{attribute 'reflection'}
FUNCTION_BLOCK FB_DevKL5151 EXTENDS FB_DevBase IMPLEMENTS iCounter
VAR_INPUT
	bInitAsCounterCard	: BOOL := FALSE; // (Default = FALSE) Use Terminal as encoder input (FALSE) or counter (TRUE) 
END_VAR
VAR CONSTANT // register values 
	WRITE_FEATURE_REGISTER 	: USINT := 16#E0; // write to register address command
	READ_FEATURE_REGISTER	: USINT := 16#A0; // Read feature register response  
END_VAR
VAR // Inputs and outputs
	Status		AT%I* : USINT ; // status byte from card
	Counter		AT%I* : UDINT ; // 
	Ctrl 		AT%Q* : USINT ; // Control byte to card`
	DataOut 	AT%Q* : UDINT ; // Set counter value
END_VAR
VAR // steppers
	InitStep : INT := 0; // init stepper
END_VAR
VAR // Manual control
	stManualControl : st_ManualCounterControl;
END_VAR

SUPER^();

METHOD PUBLIC CmdManual : BOOL
bCmdManual := TRUE;
stManualControl.nCount := Counter;

IF stManualControl.bManSetValue THEN 
	// set counter to value
	DataOut	:= stManualControl.nManValue	;
	Ctrl.2 	:= Counter <> stManualControl.nManValue;
	
	stManualControl.bManSetValue R= Counter = stManualControl.nManValue;
END_IF
END_METHOD

METHOD CmdReset : BOOL
VAR_INPUT
END_VAR
Ctrl.2 	:= FALSE;

CmdReset := NOT Status.2;
END_METHOD

METHOD CmdResetValue : BOOL // Reset the value of the counter card to 0
// set counter value to 0
DataOut	:= 0	;
Ctrl.2 	:= Counter <> 0;

CmdResetValue := Counter = 0;
END_METHOD

METHOD PUBLIC CmdSetValue : BOOL // Set the value of the counter card
VAR_INPUT
	Value	: UDINT;
END_VAR
// set counter to value
DataOut	:= Value	;
Ctrl.2 	:= Counter <> Value;

CmdSetValue := Counter = Value;
END_METHOD

PROPERTY PUBLIC CountValue : UDINT
GET
CountValue := Counter;
END_GET
END_PROPERTY

METHOD PUBLIC Init : BOOL
VAR_INPUT
	// Message location data
	nId				: UINT ; // Identification number of object
	nParentId		: UDINT ; // Id of higher level If aplicable (0 = no parent)
END_VAR

IF bInitAsCounterCard THEN
//	{warning 'Counter function needs to be added to devices'}
	ExecIdentifyDevice(nId := nId, nParentId := nParentId, eComponentType := E_ComponentTypes.NA);
ELSE 
	ExecIdentifyDevice(nId := nId, nParentId := nParentId, eComponentType := E_ComponentTypes.Encoder);
END_IF

eDevType := E_Devices.KL5151;

// Check feature register against set function 
CASE InitStep OF 
	0: // check active feature register values
		Ctrl := READ_FEATURE_REGISTER;
		InitStep := initstep + 1;
	1: // Check if operation mode is correct If not set operation mode
		IF Status = READ_FEATURE_REGISTER THEN
			//Check if we are the requested mode
			IF Counter.15 = bInitAsCounterCard THEN 
				InitStep := 3;
			ELSE
				//Copy the current value into the output
				DataOut := Counter;
				//Set the encoder/counter bit as requested
				DataOut.15 := bInitAsCounterCard;
				//Give the command to write to the card
				Ctrl := WRITE_FEATURE_REGISTER;
				InitStep := 2;
			END_IF
		END_IF
	2: // Check if register was written	
		IF Status = READ_FEATURE_REGISTER THEN
			InitStep := 3;
		END_IF
		
	3: //Stop register access, return to normal
		//Copy the current value into the output
		Ctrl := Status;
		//Reset the register access bit
		Ctrl.7 := FALSE;
		InitStep := 4;
		
	4: //Check if the command was accepted
		IF Status.7 = 0 THEN
			InitStep := 10;
		END_IF
		
	10: // init done
		bInitOk := TRUE;
		
	ELSE
		;
END_CASE

Init := bInitOk;
END_METHOD

END_FUNCTION_BLOCK

(* stored: Version 1.1.0.1, ProductVersion 3.1.4024.11
   POU FB_DevKL5151: Id {df645e77-ad73-00ed-1f06-f5798d21983d}, SpecialFunc None
   Folder Public: Id {ba5eeb51-f519-0b9d-3b18-512a69522b3c}
   Method CmdManual: Id {2c4682fb-4abf-0dcb-304c-7d205ffb993f}
   Method CmdReset: Id {1177881d-8cd4-0a69-1822-d089e6fc248e}
   Method CmdResetValue: Id {878eab4b-2982-059c-334a-891ab33aca94}
   Method CmdSetValue: Id {7a4118c4-5747-0bc6-1b86-84f27a3800c8}
   Property CountValue: Id {00e066e9-3663-0599-3e6b-d6b437f2479b}
   Get Get: Id {1e405d11-da5b-0d46-2f10-7c8c72afaea0}
   Method Init: Id {bd4538ad-b516-00fd-2eeb-cad656d156dc} *)
